// TIA Portal V20 export
VAR_GLOBAL   // PLC tag table "F-Digital_Outputs"
   FDQ_StopContactor AT %Q1200.0 : Bool;
   FDQ_LaserContactor AT %Q1200.1 : Bool;
   FDQ_LaserValidation AT %Q1200.2 : Bool;
   FDQ_FrontDoorLock AT %Q1200.3 : Bool;
   FDQ_BW_LoaderEstopRelay AT %Q1206.0 : Bool;
   FDQ_SonplasDoorClosedRelay AT %Q1206.1 : Bool;
   FDQ_FreeQ1206_2 AT %Q1206.2 : Bool;
   FDQ_FreeQ1206_3 AT %Q1206.3 : Bool;
END_VAR
